(*~
    <docu>
        <summary>
            Provides basic momentary on function.
            <para>
                To get the actual state of the momentary task, <see cref="PlcDocu.TcoCore.TcoMomentaryTask.IsOn()"/>, <see cref="PlcDocu.TcoCore.TcoMomentaryTask.IsOff()"/> and <see cref="PlcDocu.TcoCore.TcoMomentaryTask.State()"/> properties are available.
            </para>
        </summary>
    </docu>
~*)
{attribute addProperty StateOnDesc "<#On#>"}
{attribute addProperty StateOffDesc "<#Off#>"}
FUNCTION_BLOCK TcoMomentaryTask EXTENDS TcoObject IMPLEMENTS ITcoMomentaryTask
VAR
    {attribute clr [ReadOnly()]}
    _state : BOOL;
    (*~
    <docu>
        <summary>
            Use to set the state to the '''TRUE''' value.
        </summary>
    </docu>
~*)
    {attribute addProperty Name "<#Set on request#>"}
    _setOnRequest : BOOL;
    (*~
    <docu>
        <summary>
            Use to determine if the manipulation is enabled for example from the HMI application.
            This value is read only, to modify it use the property <see cref="PlcDocu.TcoCore.TcoMomentaryTask.Enabled()"/>
        </summary>
    </docu>
~*)
    {attribute addProperty Name "<#Enabled#>"}
    {attribute clr [ReadOnly()]}
    _enabled : BOOL := TRUE;
    {attribute 'hide'}
    _StartCycleCount : ULINT;
    (*~
    <docu>
        <summary>
            Indicated whether the task is in serviceable state. The default state 'serviceable' that means that the task
            can be invoked from the higher-level application. The serviceable state is cancelled when the immediate parent is `ITcoServiceable`
            and at the same time the parent is not in servicebable state. `TcoComponent` is serviceable, in order for the component's task to be
            invokable from higher-level application component must call `Service` method to induce the component into serviceable state.
        </summary>
    </docu>
    ~*)
    {attribute addProperty Name "<#Serviceable#>"}
    {attribute clr [ReadOnly()]}
    {attribute clr [RenderIgnore()]}
    _isServiceable : BOOL;
END_VAR

(*~
    <docu>
        <summary>
            Gets the context of this object.
            This context is given by declaration, its value is assigned after download by calling the implicit method <c>FB_init()</c> and cannot be changed during runtime.
        </summary>
    </docu>
~*)
PROPERTY Context : ITcoContext
GET
Context := THIS^.Parent.Context;
END_GET
END_PROPERTY

(*~
    <docu>
        <summary>
            Gets whether the any manipulation with this instance is enabled.
            The change state could be triggered with <see cref="PlcDocu.TcoCore.TcoMomentaryTask.On()"/> or <see cref="PlcDocu.TcoCore.TcoMomentaryTask.Off()"/> method call only when this property si '''TRUE'''.
        </summary>
    </docu>
~*)
PROPERTY Enabled : BOOL
GET
Enabled := _enabled;
END_GET
SET
_enabled := Enabled;

IF NOT _enabled THEN
    _state := FALSE;
    _setOnRequest := FALSE;
END_IF
END_SET
END_PROPERTY

(*~
    <docu>
        <summary>
            Gets identity of this instance.
            This value is assigned after download by calling the implicit method <c>FB_init()</c> and cannot be changed during runtime.
            This variable is used in the higher level applications.
        </summary>
    </docu>
~*)
PROPERTY Identity : ULINT
GET
Identity := _Identity;
END_GET
END_PROPERTY

PROPERTY IsOff : BOOL
GET
IsOff := NOT _state;
END_GET
END_PROPERTY

PROPERTY IsOn : BOOL
GET
IsOn := _state;
END_GET
END_PROPERTY

(*~
    <docu>
        <summary>
            Use to set the state of the '''TcoMomentaryTask''' to the value '''FALSE'''.
        </summary>
    </docu>
~*)
METHOD FINAL Off : BOOL
Off := FALSE;

//Check if Run method is called cyclically
IF THIS^.Context.StartCycleCount > _StartCycleCount + 1 THEN
    THIS^.Messenger.Programming('Run() method is not called cyclically.');
    RETURN;
END_IF

IF _state THEN
    THIS^._state := FALSE;
    OnFtrig();
    OnStateChange();
    Off := TRUE;
END_IF;
END_METHOD

(*~
    <docu>
        <summary>
            Use to set the state of the '''TcoMomentaryTask''' to the value '''TRUE'''.
        </summary>
    </docu>
~*)
METHOD FINAL On : BOOL
On := FALSE;

//Check if Run method is called cyclically
IF THIS^.Context.StartCycleCount > _StartCycleCount + 1 THEN
    THIS^.Messenger.Programming('Run() method is not called cyclically.');
    RETURN;
END_IF

IF _enabled THEN
    IF NOT _state THEN
        THIS^._state := TRUE;
        OnRtrig();
        OnStateChange();
        On := TRUE;
    END_IF;
ELSE
    THIS^.Messenger.Post('Toggletask cannot be set to TRUE as its Enabled property is FALSE.', eMessageCategory.Info);
END_IF
END_METHOD

(*~
    <docu>
        <summary>
            Executes when momentary task changes its state from '''TRUE''' to '''FALSE'''.
        </summary>
    </docu>
~*)
METHOD PROTECTED OnFtrig
END_METHOD

(*~
    <docu>
        <summary>
            Executes when momentary task changes its state from '''FALSE''' to '''TRUE'''.
        </summary>
    </docu>
~*)
METHOD PROTECTED OnRtrig
END_METHOD

(*~
    <docu>
        <summary>
            Executes when momentary task changes its state .
        </summary>
    </docu>
~*)
METHOD PROTECTED OnStateChange
END_METHOD

(*~
    <docu>
        <summary>
            This method needs to be called cyclically.
        </summary>
    </docu>
~*)
METHOD Run
VAR
    _serviceableParent : ITcoServiceable;
END_VAR
// Store the context start cycle. Used to detect if Run() method is called cyclically.
_StartCycleCount := THIS^.Context.StartCycleCount;

// Detects if parent is in serviceable state to enable manual invoke of the task from the HMI/SCADA system.
IF (THIS^.Parent <> 0) THEN
    _isServiceable := TRUE;

    IF (__QUERYINTERFACE(THIS^.Parent, _serviceableParent)) THEN
        IF (NOT _serviceableParent.IsService) THEN
            THIS^._setOnRequest := FALSE;
            _isServiceable := FALSE;
        END_IF
    END_IF
END_IF;

IF (THIS^._setOnRequest) THEN
    THIS^.On();
ELSE
    THIS^.Off();
END_IF;

IF _state THEN
    TaskOn();
ELSE
    TaskOff();
END_IF
END_METHOD

(*~
    <docu>
        <summary>
            Gets actual value of this instance.
        </summary>
    </docu>
~*)
PROPERTY State : BOOL
GET
State := _state;
END_GET
END_PROPERTY

(*~
    <docu>
        <summary>
            Executes when momentary task is in ```Off``` state .
        </summary>
    </docu>
~*)
METHOD PROTECTED TaskOff
END_METHOD

(*~
    <docu>
        <summary>
            Executes when momentary task is in  ```On``` state .
        </summary>
    </docu>
~*)
METHOD PROTECTED TaskOn
END_METHOD

END_FUNCTION_BLOCK

(* stored: Version 1.1.0.1
   POU TcoMomentaryTask: Id {2b3dea90-2b25-0f42-3297-e3bc662ebad1}, SpecialFunc None
   Property Context: Id {2a6ccb7c-f160-0d4f-387c-0fc36bf3f46f}
   Get Get: Id {a9eff097-c6d4-0344-309d-4b7dae3c6476}
   Property Enabled: Id {9ccbd869-272e-0374-0e03-3c8f2fa01c48}
   Get Get: Id {ea0810cf-22bb-017e-04e2-da10d5d8e77f}
   Set Set: Id {eea2b287-52cf-0c28-2b49-c1e3d9646357}
   Property Identity: Id {5ac2e2d0-3c45-0329-2a94-30acf57b113b}
   Get Get: Id {4c2fa687-cf31-083e-010f-c28282b5388b}
   Property IsOff: Id {c132a165-edd0-061d-357a-4338c9cae036}
   Get Get: Id {60777fb2-4bf8-0cae-0335-5802f806dcb8}
   Property IsOn: Id {4fa9c946-06c4-0807-0847-0b32d5e4a4c5}
   Get Get: Id {74954e2d-05fb-029a-0513-39c70bace59a}
   Method Off: Id {af1963cb-362b-017a-1f9f-85ae38088c9c}
   Method On: Id {b542268f-1c1c-0a1a-3094-f6ca0e1ef17f}
   Method OnFtrig: Id {7156b8d0-084a-02c1-2280-68f2b9f5ad68}
   Method OnRtrig: Id {1231dc37-77af-0405-20a9-1846142e46fd}
   Method OnStateChange: Id {96562705-edcb-005a-0da0-03cd0433d2f6}
   Method Run: Id {9839f195-c5a9-0f25-38cb-f178c6fcb458}
   Property State: Id {a9c54a34-d309-0954-2a7e-881f5102e28b}
   Get Get: Id {88b2fb9c-234f-05ca-3da0-5dd67cca05c1}
   Method TaskOff: Id {38cdf4ca-06cb-015c-10a4-b69572e4f6ae}
   Method TaskOn: Id {583d4a4a-bbd3-0518-2104-d436fac86c7a} *)
